// TIA Portal V21 export
VAR_GLOBAL   // PLC tag table "UnitàDiMisura_Codici"
END_VAR
VAR_GLOBAL CONSTANT   // user constants
   Um_Codice_m3h : DInt := 050105;
   "Um_Codice_l/m" : DInt := 050205;
   "Um_Codice_°C" : DInt := 030105;
   Um_Codice_Percentuale : DInt := 040105;
   Um_Codice_Bar : DInt := 060105;
   "Um_Codice_l/h" : DInt := 050206;
   Um_Codice_MilliBar : DInt := 060102;
END_VAR
